(* PLC project passing_sensor2, Dassault Systèmes ControlBuild 2024x Refresh1 *)
(* stored: creationDateTime 2024-01-24T08:24:06-01:00 *)

CONFIGURATION passing_sensor2
  VAR_GLOBAL
    simuperiod : REAL := 50000.0;
    taskname : STRING(50) := 'passing_sensor2.exe';
    allowpreconditions : BOOL := true;
    allowpostconditions : BOOL := true;
    status_act_prod : DINT := 0;
    m11 : REAL := 1.0;
    m12 : REAL := 0.0;
    m13 : REAL := 0.0;
    m14 : REAL := 0.0;
    m21 : REAL := 0.0;
    m22 : REAL := 1.0;
    m23 : REAL := 0.0;
    m24 : REAL := 0.0;
    m31 : REAL := 0.0;
    m32 : REAL := 0.0;
    m33 : REAL := 1.0;
    m34 : REAL := 0.0;
    m41 : REAL := 0.0;
    m42 : REAL := 0.0;
    m43 : REAL := 0.0;
    m44 : REAL := 1.0;
  END_VAR
END_CONFIGURATION
